PROGRAM MAIN
VAR
	test : TeknicEIP;
	
	ready : BOOL;
	
	contUp : BOOL;
	contDown : BOOL;
	target : REAL := -1;
END_VAR

test.bEnable := TRUE;

IF NOT ready THEN
	ready := test.homingSequence();
	RETURN;
END_IF

test.stop();
IF contUp THEN
	test.moveContinuous(direction := MC_Positive_Direction);
	contDown := FALSE;
END_IF

IF contDown THEN
	test.moveContinuous(direction := MC_Negative_Direction);
	contUp := FALSE;
END_IF


IF target >= 0 THEN
	test.moveAbsolute(targetPos := target);
	//target := 0;
END_IF


IF test.innerLimit THEN
	contDown := FALSE;
END_IF
IF test.home THEN
	contUp := FALSE;
END_IF


test();

END_PROGRAM

(* stored: Version 1.1.0.1, ProductVersion 3.1.4024.11
   POU MAIN: Id {baf0439a-1535-4c78-b2c4-6521dfd3030e}, SpecialFunc None *)
